// TIA Portal project "4m-2_V16" (V16)

(* hardware
DEVICE "S7-1200 station_1"  S7-1200 Station
   slot 0: "Rack_0"  S7-1200 Rack  Rack  V1.0
   slot 1: "PLC_1"  CPU 1212C AC/DC/Rly  6ES7 212-1BE40-0XB0  V4.2
*)

// ===== PLC "PLC_1"  CPU 1212C AC/DC/Rly =====

VAR_GLOBAL   // PLC tag table "Default tag table"
   "start" AT %I0.0 : Bool;
   "stop" AT %I0.1 : Bool;
   "M1" AT %Q0.0 : Bool;
   "M2" AT %Q0.1 : Bool;
   "X" AT %M0.0 : Bool;
   "C1" AT %M0.1 : Bool;
   "T1ON" AT %M0.2 : Bool;
   "C2" AT %M0.3 : Bool;
   "Tag_1" AT %M3.7 : Bool;
   "M2ON" AT %M0.4 : Bool;
   "cc" AT %M0.5 : Bool;
   "T2on" AT %M0.6 : Bool;
   "t2off" AT %M0.7 : Bool;
   "T3on" AT %M1.0 : Bool;
   "Tag_2" AT %M2.0 : Bool;
END_VAR

// folder: System blocks/Program resources

DATA_BLOCK "T1"   // DB1
{ S7_Optimized_Access := 'TRUE' }
AUTHOR : Simatic
FAMILY : IEC
NAME : IEC_TMR
VERSION : 1.0
// stored: InstanceOfName IEC_TIMER
"IEC_TIMER"
BEGIN
END_DATA_BLOCK

DATA_BLOCK "T2"   // DB2
{ S7_Optimized_Access := 'TRUE' }
AUTHOR : Simatic
FAMILY : IEC
NAME : IEC_TMR
VERSION : 1.0
// stored: InstanceOfName IEC_TIMER
"IEC_TIMER"
BEGIN
END_DATA_BLOCK

DATA_BLOCK "timer3"   // DB3
{ S7_Optimized_Access := 'TRUE' }
AUTHOR : Simatic
FAMILY : IEC
NAME : IEC_TMR
VERSION : 1.0
// stored: InstanceOfName IEC_TIMER
"IEC_TIMER"
BEGIN
END_DATA_BLOCK

// folder: (top level)

ORGANIZATION_BLOCK "Main"   // OB1, LAD, ProgramCycle
TITLE = "Main Program Sweep (Cycle)"
{ S7_Optimized_Access := 'TRUE' }
VERSION : 0.1
   VAR_INPUT
      Initial_Call : Bool;   // Initial call of this OB
      Remanence : Bool;   // =True, if remanent data are available
   END_VAR
   VAR_TEMP   // added for the SCL form of the ladder/FBD networks
      _w1 : Bool;
   END_VAR
BEGIN

REGION Network 1
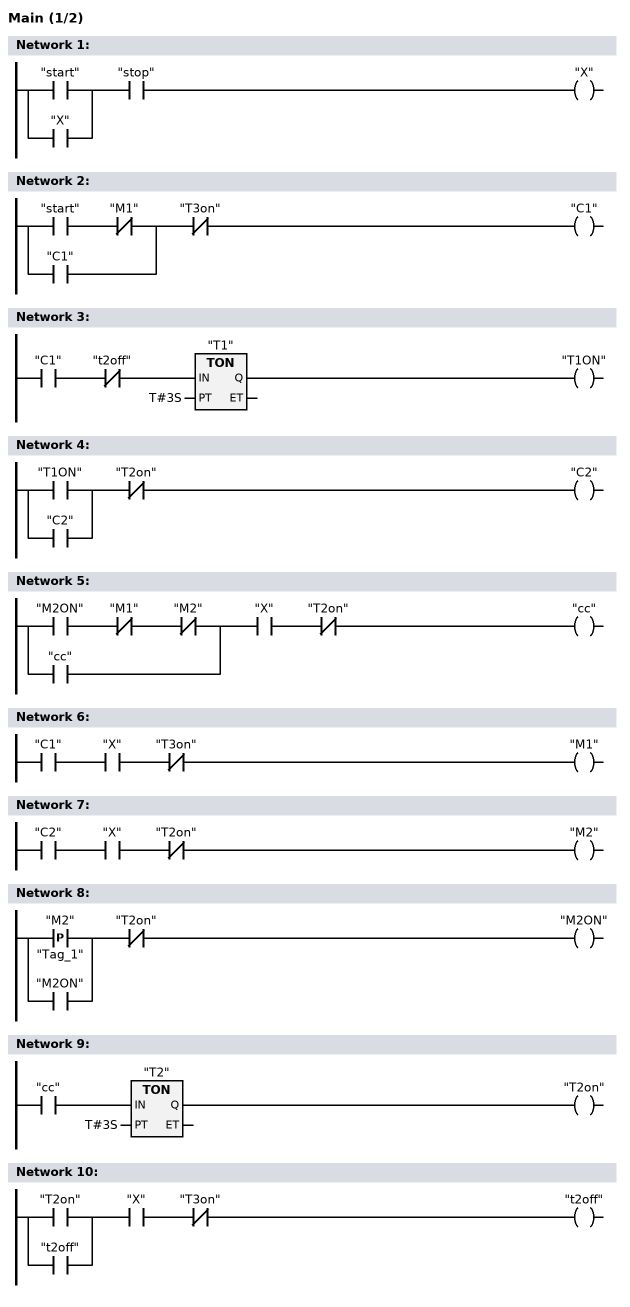
   RUNG wire#powerrail
      Contact( "start" )
      wire#w1
      Contact( "stop" )
      Coil( "X" )
   END_RUNG
   RUNG wire#powerrail
      Contact( "X" )
   END_RUNG wire#w1
   // the same network as SCL:
   "X" := ("start" OR "X") AND "stop";
END_REGION

REGION Network 2
   RUNG wire#powerrail
      Contact( "start" )
      I_Contact( "M1" )
      wire#w1
      I_Contact( "T3on" )
      Coil( "C1" )
   END_RUNG
   RUNG wire#powerrail
      Contact( "C1" )
   END_RUNG wire#w1
   // the same network as SCL:
   "C1" := (("start" AND NOT "M1") OR "C1") AND NOT "T3on";
END_REGION

REGION Network 3
   "T1".TON(IN := "C1" AND NOT "t2off", PT := T#3S);
   "T1ON" := "T1".Q;
END_REGION

REGION Network 4
   RUNG wire#powerrail
      Contact( "T1ON" )
      wire#w1
      I_Contact( "T2on" )
      Coil( "C2" )
   END_RUNG
   RUNG wire#powerrail
      Contact( "C2" )
   END_RUNG wire#w1
   // the same network as SCL:
   "C2" := ("T1ON" OR "C2") AND NOT "T2on";
END_REGION

REGION Network 5
   RUNG wire#powerrail
      Contact( "M2ON" )
      I_Contact( "M1" )
      I_Contact( "M2" )
      wire#w1
      Contact( "X" )
      I_Contact( "T2on" )
      Coil( "cc" )
   END_RUNG
   RUNG wire#powerrail
      Contact( "cc" )
   END_RUNG wire#w1
   // the same network as SCL:
   "cc" := (("M2ON" AND NOT "M1" AND NOT "M2") OR "cc") AND "X" AND NOT "T2on";
END_REGION

REGION Network 6
   RUNG wire#powerrail
      Contact( "C1" )
      Contact( "X" )
      I_Contact( "T3on" )
      Coil( "M1" )
   END_RUNG
   // the same network as SCL:
   "M1" := "C1" AND "X" AND NOT "T3on";
END_REGION

REGION Network 7
   RUNG wire#powerrail
      Contact( "C2" )
      Contact( "X" )
      I_Contact( "T2on" )
      Coil( "M2" )
   END_RUNG
   // the same network as SCL:
   "M2" := "C2" AND "X" AND NOT "T2on";
END_REGION

REGION Network 8
   RUNG wire#powerrail
      P_Contact(operand := "M2", bit := "Tag_1")
      wire#w1
      I_Contact( "T2on" )
      Coil( "M2ON" )
   END_RUNG
   RUNG wire#powerrail
      Contact( "M2ON" )
   END_RUNG wire#w1
   // the same network as SCL:
   #_w1 := "M2" AND NOT "Tag_1";   // rising edge of "M2"
   "Tag_1" := "M2";
   "M2ON" := (#_w1 OR "M2ON") AND NOT "T2on";
END_REGION

REGION Network 9
   "T2".TON(IN := "cc", PT := T#3S);
   "T2on" := "T2".Q;
END_REGION

REGION Network 10
   RUNG wire#powerrail
      Contact( "T2on" )
      wire#w1
      Contact( "X" )
      I_Contact( "T3on" )
      Coil( "t2off" )
   END_RUNG
   RUNG wire#powerrail
      Contact( "t2off" )
   END_RUNG wire#w1
   // the same network as SCL:
   "t2off" := ("T2on" OR "t2off") AND "X" AND NOT "T3on";
END_REGION

REGION Network 11
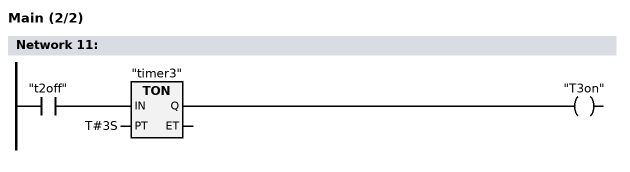
   "timer3".TON(IN := "t2off", PT := T#3S);
   "T3on" := "timer3".Q;
END_REGION
END_ORGANIZATION_BLOCK